# B&R Automation Studio project CamAutomat1 (part 2)

#### Main.st
```iecst
//[*********************************************************************************
//* Primary Author:    	Morteza Shahmoradi
//* Created:   			Dec 4, 2023
//* Description: 		Machine  Control
//	*********************************************************************************]
PROGRAM _INIT

	(* Initialize MpAxisBasic_AxisMaster *)
	MpAxisBasic_AxisMaster.Enable := TRUE;
	AxisParameters_Master.Position := 0.0;
	AxisParameters_Master.Velocity := 72.0;
	AxisParameters_Master.Acceleration := 3600.0;
	AxisParameters_Master.Deceleration := 3600.0;
	AxisParameters_Master.Jog.Deceleration := 3600;
	AxisParameters_Master.Stop.Deceleration := 3600.0;
	(* Initialize MpAxisBasic_AxisSlave *)
	MpAxisBasic_AxisSlave.Enable := TRUE;
	AxisParameters_Slave.Position := 0.0;
	AxisParameters_Slave.Velocity := 72.0;
	AxisParameters_Slave.Acceleration := 3600.0;
	AxisParameters_Slave.Deceleration := 3600.0;
	AxisParameters_Slave.Stop.Deceleration := 3600.0;
	AxisParameters_Slave.Jog.Deceleration := 3600;
	AxisParameters_Slave.Stop.Deceleration := 3600.0;

	AxisParameters_Master.AutoTune.Mode 				:= mcAXIS_TUNE_AUTOMATIC;
	AxisParameters_Master.AutoTune.MaxCurrentPercent 	:= 80.0;
	AxisParameters_Master.AutoTune.MaxDistance 			:= 10;
	AxisParameters_Master.AutoTune.MaxPositionError 	:= 30;

	AxisParameters_Slave.AutoTune.Mode 				:= mcAXIS_TUNE_AUTOMATIC;
	AxisParameters_Slave.AutoTune.MaxCurrentPercent 	:= 80.0;
	AxisParameters_Slave.AutoTune.MaxDistance 			:= 10;
	AxisParameters_Slave.AutoTune.MaxPositionError 	:= 30;

	MpAxisBasic_AxisMaster.MpLink := ADR(gConv_MpLink);
	MpAxisBasic_AxisMaster.Parameters := ADR(AxisParameters_Master);
	MpAxisBasic_AxisSlave.MpLink := ADR(gCutter_MpLink);
	MpAxisBasic_AxisSlave.Parameters := ADR(AxisParameters_Slave);
	MpAxisCamSequencer_0.MpLink := ADR(gCutter_MpLink);

	MpAxisCamSequencer_0.MpLinkMaster := ADR(gConv_MpLink);
	MpAxisCamSequencer_0.Parameters := ADR(CamSequencerParameters_0);

END_PROGRAM

PROGRAM _CYCLIC

	AxisParameters_Master.Velocity := gConvPrSpeed * 70 / 60 ;	// speed comes the part per minites divided by 60 s
	AxisParameters_Slave.Jog.Velocity := gCutJogSpeed;	  // Jog speed comes from HMi manaul page
	AxisParameters_Master.Jog.Velocity := gConvJogSpeed; // belt jog peed  comes from HMi manaul page
	gConvPosition := MpAxisBasic_AxisMaster.Position;  // realtime belt position  to  HMi manaul page
	gCutPosition  := MpAxisBasic_AxisSlave.Position;  // real time saw position to hmi
	gManualActive :=  NOT MpAxisBasic_AxisMaster.MoveVelocity;
	IF  (MpAxisBasic_AxisSlave.Position < cutJogEnableFWL) THEN // if the saw is not in cut zone move is backward
		AxisParameters_Slave.Direction := mcDIR_NEGATIVE;
	ELSE
		AxisParameters_Slave.Direction :=  mcDIR_POSITIVE;

	END_IF
	// Check the saw to  find where is connected
	sawInCutPosition := NOT (MpAxisBasic_AxisSlave.Position > cutJogEnableBWL AND MpAxisBasic_AxisSlave.Position < cutJogEnableFWM) AND NOT MpAxisBasic_AxisMaster.MoveVelocity ;
	displayMessageAuto := NOT sawInCutPosition AND NOT MpAxisBasic_AxisMaster.MoveVelocity ; // dispay disable message so no possibe run
	TON_DelayDo1.PT := DelayOpc;

	// Create Pulse Generator Start
	IF TON_DelayDo1.ET <> DelayOpc THEN
		TON_DelayDo1.IN := TRUE;
	END_IF
	TON_DelayDo1();
	gServoInitialized:= TON_DelayDo1.Q ;
	gDispalyServoNotReady := NOT gServoInitialized;

	// Control and Case for the Cutter and Conveyor
		CASE AxisStep OF

				STATE_WAIT :     // Wait until servo initialized  00000 ************************** STATE_WAIT ********************* 0000 ********************* STATE_WAIT
					MpAxisBasic_AxisMaster.Power		:= FALSE; // turn of drive
					MpAxisBasic_AxisSlave.Power			:= FALSE; // turn of drive Saw
					MpAxisCamSequencer_0.Enable			:= FALSE; // diale the cam sequencer
					gEnableTouchProbe := FALSE;
					IF ( Axis1.Exists AND gServoInitialized) THEN
						MpAxisBasic_AxisMaster.Power	:= TRUE;
						MpAxisBasic_AxisSlave.Power		:= TRUE;
						AxisStep :=  STATE_POWER_ON;
					END_IF

				STATE_POWER_ON : //Power on the servos **** 1 ****************** STATE_POWER_ON ********************* 1 ********************* STATE_POWER_ON
					gEnableTouchProbe := FALSE;
					IF (MpAxisBasic_AxisMaster.PowerOn = TRUE AND MpAxisBasic_AxisMaster.PowerOn = TRUE ) THEN
						AxisStep := STATE_HOME;
					END_IF
					IF (MpAxisBasic_AxisMaster.Error OR MpAxisBasic_AxisSlave.Error) THEN
						Axis1_ErrorID := 1;
						AxisStep := STATE_ERROR;
					END_IF

				STATE_HOME :  //Home the two Servo ********* 2 ********************STATE_HOME************************* 2 *********************STATE_HOME
					Axis1.statusHomed 							:= FALSE;
					AxisParameters_Master.Homing.Mode 		:= mcHOMING_DIRECT;// set the home type for the master ax
					AxisParameters_Master.Homing.Position 	:= 0.0;
					AxisParameters_Slave.Homing.Mode 		:= mcHOMING_ABSOLUTE; // set the home type abs for the slave
					AxisParameters_Slave.Homing.Position 	:= -161.4;  // relative position
					IF (NOT MpAxisCamSequencer_0.CommandBusy AND NOT MpAxisCamSequencer_0.StartSequence)  THEN
						MpAxisBasic_AxisMaster.Home 			:= TRUE;
						MpAxisBasic_AxisSlave.Home 			:= TRUE;
					END_IF

					IF EDGEPOS(MpAxisBasic_AxisMaster.IsHomed) THEN // master is homed
						Axis1Home		:= TRUE;
					END_IF

					IF EDGEPOS(MpAxisBasic_AxisSlave.IsHomed) THEN // slave is homed
						Axis2Home		:= TRUE;
					END_IF

					IF (Axis1Home AND Axis2Home) THEN  // if its home then go to ready state
						Axis1.statusHomed 			:= 1;
						MpAxisBasic_AxisMaster.Home 	:= FALSE;
						MpAxisBasic_AxisSlave.Home 	:= FALSE;
						Axis2Home := FALSE;
						Axis1Home := FALSE;
						MpAxisCamSequencer_0.Enable := TRUE;
						gEnableTouchProbe := TRUE;
						AxisStep := STATE_READY;
					END_IF
					IF (MpAxisBasic_AxisMaster.Error OR MpAxisBasic_AxisSlave.Error) THEN  // if there is an erro o to error state
						Axis1_ErrorID := 2;
						AxisStep := STATE_ERROR;
					END_IF

				STATE_READY : //Wait for the commands to change the state ***** 10 ************************ STATE_READY ******************** 10 ************************** STATE_READY
					Axis1.statusOff := 0;
					Axis1.statusStarting :=0;
					MpAxisCamSequencer_0.Enable := TRUE;
					gEnableTouchProbe := FALSE;
					CutStart := FALSE;
					disbaleHome := TRUE;	// Enable home
						// Home state if requested by HMI
					IF (Axis1.cmdHome = 1 AND NOT  MpAxisBasic_AxisMaster.CommandBusy  AND NOT  MpAxisBasic_AxisSlave.CommandBusy )THEN  // command home if
						Axis1Home							:= FALSE;
						Axis2Home							:= FALSE;
						MpAxisCamSequencer_0.StartSequence 	:= FALSE;
						AxisStep 							:= STATE_HOME;
						Axis1.cmdHome		 				:= FALSE;

					ELSIF (Axis1.cmdStop = 1) THEN  // Stop command activate from HMI

						Axis1.cmdCamAutomat 					:=FALSE;
						Axis1.cmdStop 							:= FALSE;
						Axis1.cmdMoveVelocity 					:= FALSE;
						Axis1.cmdMoveAdditive 					:= FALSE;
						MpAxisBasic_AxisMaster.MoveAdditive 	:= FALSE;
						MpAxisBasic_AxisMaster.MoveVelocity 	:= FALSE;
						AxisStep 				:= STATE_STOP;

					ELSIF MpAxisBasic_AxisMaster.MoveVelocity AND Axis1.cmdStartAutomat   THEN  // demand for the Cut
						MpAxisCamSequencer_0.StartSequence := TRUE;
						MpAxisCamSequencer_0.Signal1		:= FALSE;
						AxisStep := STATE_MOVE_CAMAUTOMAT;

					ELSIF NOT MpAxisBasic_AxisSlave.MoveAbsolute AND Axis1.cmdMoveVelocity AND NOT MpAxisBasic_AxisMaster.MoveVelocity AND  MpAxisBasic_AxisSlave.Position = 0.0  THEN
							AxisStep := STATE_MOVE_VELOCITY;
					ELSIF Axis1.cmdMoveVelocity  AND NOT (MpAxisBasic_AxisSlave.Position = 0.0  ) THEN
						MpAxisBasic_AxisSlave.MoveAbsolute := TRUE;
					ELSIF MpAxisBasic_AxisSlave.MoveAbsolute  AND  ( MpAxisBasic_AxisSlave.Position = 0.0 ) THEN
						MpAxisBasic_AxisSlave.MoveAbsolute := FALSE;
					ELSIF Axis2.cmdHome THEN
						MpAxisBasic_AxisSlave.MoveAbsolute := TRUE;
						Axis2.cmdHome := FALSE;
					ELSIF NOT MpAxisBasic_AxisMaster.MoveVelocity AND (Axis1.cmdManualForward OR Axis1.cmdManualReverse OR Axis2.cmdManualForward OR Axis2.cmdManualReverse ) THEN
						AxisStep := STATE_JOG;
						startPositionJog := MpAxisBasic_AxisMaster.Position ;
					ELSIF (Axis1.Exists = 0) THEN  // power of servos
						AxisStep := STATE_WAIT;

					END_IF

					IF MpAxisBasic_AxisMaster.Error OR MpAxisBasic_AxisSlave.Error THEN  // if there is an erro o to error state
						AxisStep := STATE_ERROR;
					END_IF

				STATE_STOP : // Stop the axis ******** 20 ****************************** STATE_STOP ***************************** 20 ********************** STATE_STOP
					Axis1.statusOff := 0;
					MpAxisBasic_AxisMaster.Stop := TRUE;
					MpAxisBasic_AxisSlave.Stop := TRUE;
					(* if axis is stopped go to state wait *)
					IF (MpAxisBasic_AxisMaster.Stopped = 1 AND MpAxisBasic_AxisSlave.Stopped = 1 ) THEN
					MpAxisBasic_AxisMaster.Stop := FALSE;
					MpAxisBasic_AxisSlave.Stop := FALSE;
						AxisStep := STATE_READY;
					END_IF
					(* check if error occured *)
					IF (MpAxisBasic_AxisMaster.Error OR MpAxisBasic_AxisSlave.Error) THEN
						Axis1_ErrorID := 3;
						AxisStep := STATE_ERROR;
					END_IF
				STATE_MOVE_ABSOLUTE : //Control Move Absolute **** 24 *************************** STATE_MOVE_ABSOLUTE *********************** 24 ******************* STATE_MOVE_ABSOLUTE

				STATE_MOVE_ADDITIVE : //Control Move Additive ** 26 *********************** STATE_MOVE_POSITION *************************** 26 ****************************STATE_MOVE_POSITION
					IF ( Axis1.cmdMoveAdditive  )	 THEN
						MpAxisBasic_AxisMaster.MoveAdditive := TRUE;
						Axis1.cmdMoveAdditive := FALSE;
						TON_StepDelay.IN			:= TRUE;
						AxisStep := STATE_READY;
					END_IF

					IF MpAxisBasic_AxisMaster.Error THEN  // if there is an erro o to error state
						AxisStep := STATE_ERROR;
					END_IF

				STATE_MOVE_VELOCITY : //Control Move velocity ** 28 *************************** STATE_MOVE_VELOCITY *********************** 28 ******************* STATE_MOVE_VELOCITY
					IF ( Axis1.cmdMoveVelocity  ) 	THEN
						MpAxisBasic_AxisMaster.MoveVelocity	:= TRUE;
						Axis1.cmdMoveVelocity := FALSE;
						AxisStep := STATE_READY;
					TON_StepDelay.IN			:= TRUE;
					Axis1.cmdStartAutomat 		:= TRUE;
					END_IF

					IF MpAxisBasic_AxisMaster.Error THEN
						AxisStep := STATE_ERROR;
					END_IF

				STATE_MOVE_CAMAUTOMAT : //Control Move automat *** 30 *************************** STATE_MOVE_VELOCITY *********************** 30 ******************* STATE_MOVE_CAMAUTOMAT
						gEnableTouchProbe := TRUE;
						MpAxisBasic_AxisMaster.Update := gSaveParameter;
						MpAxisCamSequencer_0.Signal2 := Axis1.statusOff ;
						CutStart := MpAxisCamSequencer_0.ActualStateIndex <> 0 AND enableCut;
						gEnableTouchProbe := CutStart;
					 IF NOT Axis1.cmdStartAutomat  THEN  // demand for cut activate from HMI
						Axis1.cmdCam 			:= FALSE;
						MpAxisCamSequencer_0.StartSequence 		:= FALSE;
						AxisStep := STATE_READY;
					ELSIF (Axis1.cmdStop = 1) THEN
						enableCut								:= FALSE; // Enable cut will be clear as stop cmamnd comes
						Axis1.cmdStartAutomat 					:= FALSE;
						Axis1.cmdCam 							:= FALSE;
						Axis1.cmdStop 							:= FALSE;
						Axis1.cmdMoveVelocity 					:= FALSE;
						Axis1.cmdMoveAdditive 					:= FALSE;
						MpAxisBasic_AxisMaster.MoveAdditive 	:= FALSE;
						MpAxisBasic_AxisMaster.MoveVelocity 	:= FALSE;
						MpAxisCamSequencer_0.StartSequence		:= FALSE;
						AxisStep := STATE_STOP;
					ELSIF (Axis1.statusOff = 1 AND MpAxisCamSequencer_0.ActualStateIndex = 1 ) THEN
						Axis1.cmdStartAutomat 					:= FALSE;  // production finish procedure
						Axis1.cmdCam 							:= FALSE;
						Axis1.statusOff							:= FALSE;
						Axis1.cmdMoveVelocity 					:= FALSE;
						Axis1.cmdMoveAdditive 					:= FALSE;
						MpAxisBasic_AxisMaster.MoveAdditive 	:= FALSE;
						MpAxisBasic_AxisMaster.MoveVelocity 	:= FALSE;
						MpAxisCamSequencer_0.StartSequence		:= FALSE;
						AxisStep := STATE_STOP;
						enableCut								:= FALSE;
					ELSIF MpAxisCamSequencer_0.ActualStateIndex >=1 THEN
						MpAxisCamSequencer_0.Signal1 := Axis1.cmdCam AND NOT Axis1.statusOff AND NOT twoCutEnable ;
						MpAxisCamSequencer_0.Signal2 := Axis1.cmdCam AND NOT Axis1.statusOff AND  twoCutEnable ;

					END_IF

				STATE_JOG ://************************* 40 **************************** STATE_JOG ********************************* 40 ********************* STATE_JOG

				IF NOT (Axis1.cmdManualForward OR Axis1.cmdManualReverse OR Axis2.cmdManualForward OR Axis2.cmdManualReverse ) AND  gRunPage THEN
					gRunPage := FALSE;
					AxisStep := STATE_READY;
				END_IF

				MpAxisBasic_AxisMaster.JogPositive 	:= Axis1.cmdManualForward AND sawInCutPosition; // Jog Conveyor forward
				MpAxisBasic_AxisMaster.JogNegative	:= Axis1.cmdManualReverse AND MpAxisBasic_AxisMaster.Position > (startPositionJog - 100.00) AND sawInCutPosition;
				IF 	EDGENEG(Axis1.cmdManualForward) THEN // correct the position
					startPositionJog := MpAxisBasic_AxisMaster.Position;
				END_IF
				MpAxisBasic_AxisSlave.JogPositive 	:= Axis2.cmdManualForward AND cutJogEnableFW   ;// Jog Cutter Forward
				MpAxisBasic_AxisSlave.JogNegative 	:= Axis2.cmdManualReverse AND cutJogEnableBW ; // Jog Cutter Reverse
				disbaleHome := FALSE; // disable to make zero in hmi

				STATE_ERROR : //********************** 101 ******************************* STATE_ERROR **************************** 101 ********************** STATE_ERROR
					gErrorID := 3;
					alarmActive := TRUE;
					enableCut := FALSE;
					Axis1.statusStarting :=0;
					Axis1.statusFaulted := TRUE;
					MpAxisBasic_AxisMaster.Power := FALSE;
					MpAxisBasic_AxisMaster.Home := FALSE;
					MpAxisBasic_AxisMaster.Stop := FALSE;
					MpAxisBasic_AxisMaster.MoveAbsolute := FALSE;
					MpAxisBasic_AxisMaster.MoveVelocity := FALSE;
					MpAxisBasic_AxisMaster.ErrorReset := Axis1.cmdReset;
					MpAxisBasic_AxisSlave.Power := FALSE;
					MpAxisBasic_AxisSlave.Home := FALSE;
					MpAxisBasic_AxisSlave.Stop := FALSE;
					MpAxisBasic_AxisSlave.MoveAbsolute := FALSE;
					MpAxisBasic_AxisSlave.MoveVelocity := FALSE;
					MpAxisBasic_AxisSlave.ErrorReset := Axis1.cmdReset;
					MpAxisCamSequencer_0.ErrorReset := Axis1.cmdReset;
					IF (NOT(MpAxisBasic_AxisSlave.Error ) AND NOT(MpAxisBasic_AxisMaster.Error )) THEN
						Axis1.statusFaulted:=FALSE;
						Axis1.cmdReset := FALSE;
						AxisStep := STATE_WAIT;
						Axis1.statusErrorID := 0;
						MpAxisBasic_AxisMaster.ErrorReset := FALSE;
						MpAxisBasic_AxisSlave.ErrorReset  := FALSE;
					MpAxisCamSequencer_0.ErrorReset := FALSE;
					gErrorID := 0;
					alarmActive := FALSE;

					END_IF

	END_CASE
	// Graph in the C# app
	Data[0] := MpAxisBasic_AxisMaster.Position;
	Data[1] := MpAxisBasic_AxisSlave.Position;
	Data[2] := BOOL_TO_REAL(Axis1.cmdCam) * 360.0;
	Data[3] := 0.0;
	Data[4] := 0.0;
	Data[5] := MpAxisCamSequencer_0.ActualStateIndex * 50.0;
	// Call fbs
	MpAxisBasic_AxisMaster();
	MpAxisBasic_AxisSlave();
	MpAxisCamSequencer_0();
	// Stop blade pass the cut zone
	cutJogEnableFW := (MpAxisBasic_AxisSlave.Position > -0.1  AND MpAxisBasic_AxisSlave.Position < cutJogEnableFWL ) OR // stop jog when the blade is off
	(MpAxisBasic_AxisSlave.Position > cutJogEnableFWM  AND MpAxisBasic_AxisSlave.Position < 359.9999) OR
	bypassProtection;
	cutJogEnableBW := (MpAxisBasic_AxisSlave.Position > -0.1  AND MpAxisBasic_AxisSlave.Position < cutJogEnableBWL ) OR // stop jog when the blade is off
	(MpAxisBasic_AxisSlave.Position > cutJogEnableBWM  AND MpAxisBasic_AxisSlave.Position < 359.9999) OR
	bypassProtection;

	IF gErrorID > 0 THEN  // MAchine status code
		gMachineStatus := 3; // Error
		displayStopImage := TRUE;
		displayRunImage := FALSE;
	ELSIF AxisStep = 0 AND gServoInitialized  THEN
		gMachineStatus := 6;
		displayStopImage := TRUE;
		displayRunImage := FALSE;
	ELSIF MpAxisBasic_AxisMaster.MoveVelocity AND gErrorID = 0 THEN // define the stop mode
		gMachineStatus := 1;
		displayStopImage := FALSE;
		displayRunImage := TRUE;
	ELSIF AxisStep = 40 THEN
		gMachineStatus := 2;
		displayStopImage := TRUE;
		displayRunImage := FALSE;
	ELSIF Axis1.statusOff = 1 THEN // define the stop mode finalize mpod
		gMachineStatus := 5;
		displayStopImage := TRUE;
		displayRunImage := FALSE;
	ELSIF NOT MpAxisBasic_AxisMaster.MoveVelocity AND AxisStep = 10   THEN // define the Jog mode
		gMachineStatus := 0;
		displayStopImage := TRUE;
		displayRunImage := FALSE;
	ELSIF gServoInitialized = 0 THEN // servo are intialized
		gMachineStatus := 4;
		displayStopImage := TRUE;
		displayRunImage := FALSE;
	END_IF

	gMachineStatusMessage := gMachineStatusArray[gMachineStatus];	 // HMI status
	cutEnd := (MpAxisBasic_AxisSlave.Position > cutStartDegree AND MpAxisBasic_AxisSlave.Position < cutEndDegree ) OR (MpAxisBasic_AxisSlave.Position > cutStartDegree + 180.0 AND MpAxisBasic_AxisSlave.Position < cutEndDegree +180 AND twoCutEnable );
	maxproducSpeed := maxSpeed + maxSpeed * 0.855 * twoCutEnable; // max production speed
	IF gConvPrSpeed > maxproducSpeed THEN // limit the speed to prevent fault
		gConvPrSpeed := maxproducSpeed;
	END_IF

	IF EDGEPOS(cutEnd) THEN  // if one cut done cut the signal plc
		Axis1.cmdCam := FALSE;
		cutCount := cutCount +1; // add one cut is done
	END_IF

	IF gResetCount THEN  // reset cut count
		cutCount := 0;
	END_IF

END_PROGRAM

PROGRAM _EXIT

	MpAxisBasic_AxisMaster.Enable := FALSE;
	MpAxisBasic_AxisSlave.Enable := FALSE;
	MpAxisCamSequencer_0.Enable := FALSE;
	MpAxisBasic_AxisMaster();
	MpAxisBasic_AxisSlave();
	MpAxisCamSequencer_0();

END_PROGRAM
```

### Program Logical/TouchProbe (IEC) - Save position and control trigger

#### Variables.var
```iecst
VAR
	ValidTriggerCount : UDINT; (*ValidTriggerCount comes from touch probe*)
	preValue : LREAL; (*Old position*)
	partDetected : BOOL; (*start cam*)
	newValueF : BOOL; (*New Value comes form MC BR*)
	newValue : LREAL; (*new Position*)
	MissedTriggerCount : UDINT; (*MissedTriggerCount from touch robe *)
	missedCuts : INT; (*Number of missed cuts*)
	MinWidth : LREAL := 9.0; (*MinWidth to the MC BR touchprobe, to get the valid triiger*)
	MC_BR_TouchProbe_0 : MC_BR_TouchProbe := (Period:=70,ExpectedValue:=70,WindowNegative:=20,WindowPositive:=20,Mode:=mcTP_MODE_WITHOUT_PERIOD); (*MC probe to detec the position*)
	MC_BR_ProcessParID_AcpAx_0 : MC_BR_ProcessParID_AcpAx; (*Set the battery problem Par block*)
	McBrTrigger : McBrTriggerType; (*MC Br Trigger*)
	McBrAdvancePar : McAdvBrTouchProbeParType := (ReadTriggerWidth:=1); (*MC Advance paramter*)
	McAcpAxProcessParIDPar : McAcpAxProcessParIDType := (ParID:=719,VariableAddress:=1,DataType:=mcACPAX_PARTYPE_UDINT); (*parameters*)
	MaxWidth : LREAL := 11.0; (*Maximum width for the MC triiger type - touc probe*)
	maxValueExpected : LREAL := 100.00; (*MAximum Expected Value*)
	lastAndCurrentDif : LREAL; (*last and current disatnce*)
	i : USINT; (*for saving the cuts*)
	difValue : LREAL; (*distance*)
	delatTimerProbe : TON; (*Delay for start cut*)
	cutSize : LREAL := 10.0; (*Cut Size *)
	cutDistanceAveHmi : LREAL; (*Average of last cuts to be display in hmi*)
	cutDistanceAve : LREAL; (*Average of last cuts *)
	cutDistance : ARRAY[0..7] OF LREAL; (*Lat 8 cut distance*)
	MC_BR_TouchProbe_1 : MC_BR_TouchProbe := (Period:=70,ExpectedValue:=70,WindowNegative:=20,WindowPositive:=20,Mode:=mcTP_MODE_SHIFT_FROM_RESULT); (*MC probe to detec the position*)
	McBrTrigger_1 : McBrTriggerType; (*MC Br Trigger*)
	McBrAdvancePar_1 : McAdvBrTouchProbeParType := (UseFirstTriggerPosition:=1); (*MC Advance paramter*)
	MC_BR_ProcessParID_AcpAx_1 : MC_BR_ProcessParID_AcpAx; (*Set the battery problem Par block conv*)
	currentReadingDistance : LREAL; (*Reead the current distance beween two print mark*)
END_VAR
```

#### Main.st
```iecst
//[*********************************************************************************
//* Primary Author:    	Morteza Shahmoradi
//* Created:   			Dec 7, 2023
//* Description: 		Touch Probe
//	*********************************************************************************]
PROGRAM _INIT
	(* Insert code here *)

	MC_BR_TouchProbe_1.Enable := TRUE;

END_PROGRAM

PROGRAM _CYCLIC
	// Code to write the par id 719 19, to bypass the encoder alarm, for cutter
	MC_BR_ProcessParID_AcpAx_0(Axis := ADR(gCutter_MpLink), DataAddress := ADR(McAcpAxProcessParIDPar) , NumberOfParIDs :=1 , Mode := mcACPAX_PARID_SET);
	MC_BR_ProcessParID_AcpAx_0();
	MC_BR_ProcessParID_AcpAx_1(Axis := ADR(gConv_MpLink), DataAddress := ADR(McAcpAxProcessParIDPar) , NumberOfParIDs :=1 , Mode := mcACPAX_PARID_SET);
	MC_BR_ProcessParID_AcpAx_1();

	// touch probe setup,
	MC_BR_TouchProbe_0.AdvancedParameters := McBrAdvancePar;
	MC_BR_TouchProbe_0.Axis := ADR(gConv_MpLink);
	MC_BR_TouchProbe_0.TriggerInput := McBrTrigger;
	MC_BR_TouchProbe_0();
	MC_BR_TouchProbe_0.Enable := gEnableTouchProbe;

	McBrAdvancePar.ReadTriggerWidth := TRUE; // Enable to read print lengh
	ValidTriggerCount := MC_BR_TouchProbe_0.ValidTriggerCount;// count of valid trigger
	MissedTriggerCount := MC_BR_TouchProbe_0.MissedTriggerCount; // count of missed trigger
	MC_BR_TouchProbe_0.TriggerInput.MaxWidth := MaxWidth; // MaxWidth to the touch probe
	MC_BR_TouchProbe_0.TriggerInput.MinWidth := MinWidth; // Min Width to the touch rpobe

	// second touch probe for training purpose
	MC_BR_TouchProbe_1.AdvancedParameters := McBrAdvancePar_1;
	MC_BR_TouchProbe_1.Axis := ADR(gConv_MpLink);
	MC_BR_TouchProbe_1.TriggerInput := McBrTrigger_1;
	MC_BR_TouchProbe_1();
	MC_BR_TouchProbe_1.Enable := NOT gResetCount;

	currentReadingDistance := MC_BR_TouchProbe_1.Period - MC_BR_TouchProbe_1.DeltaExpectedValue;

	// manaul paramter find

	newValue := MC_BR_TouchProbe_0.RecordedValue;
	IF newValue > ( preValue + cutSize) THEN  // check if its a new print mark coms
		difValue := newValue - preValue ;  // calculates
		IF difValue > gMinValue THEN   // validate correct distance
			newValueF := TRUE;
			preValue := newValue;
			partDetected := delatTimerProbe.Q ; // part is detected rise cut flag
			IF difValue < maxValueExpected THEN
				FOR i := 0 TO 6 BY 1 DO
					cutDistance[7-i] := cutDistance[6-i] ;
				END_FOR
				cutDistance [0] := difValue;
				lastAndCurrentDif := difValue; // for Hmi display
				cutDistanceAve := 0;
				FOR i := 0 TO 7 BY 1 DO			// save old data
					cutDistanceAve := cutDistanceAve + cutDistance[i] ;
				END_FOR
				cutDistanceAveHmi := cutDistanceAve/ 8;
			END_IF
		END_IF

		IF difValue < gMinValue AND newValueF THEN   // count missed cuts
			missedCuts := missedCuts + 1;
			newValueF := FALSE;
		END_IF

	END_IF

	IF gResetCount THEN  // reset cut count
		missedCuts := 0;
		gResetCount := FALSE;
	END_IF

	delatTimerProbe(IN := CutStart , PT := T#500ms);
	delatTimerProbe();
	IF 	EDGEPOS(partDetected) AND delatTimerProbe.Q  THEN // activate the cut when the touch is 70mm after that
		Axis1.cmdCam := TRUE;
		partDetected := FALSE;
	END_IF

	IF EDGEPOS(Axis1.cmdStartAutomat) THEN // transfer the cut last and new position to the last position
		preValue := newValue;
	END_IF
	IF EDGEPOS(gEnableTouchProbe) THEN  // reset the partDetected bit to prevent stop in jog
		partDetected := FALSE;
	END_IF

	//  get paramter infor from cam automat

END_PROGRAM

PROGRAM _EXIT
	(* Insert code here *)
	MC_BR_TouchProbe_0.Enable := FALSE;
	MC_BR_TouchProbe_0();
	MC_BR_TouchProbe_1.Enable := FALSE;
	MC_BR_TouchProbe_1();

END_PROGRAM
```

### Program Logical/MachineAlarm (IEC) - Alarm Control

#### Variables.var
```iecst
VAR
	MpAlarmXCore_0 : MpAlarmXCore; (*mp alarm core x function block *)
	MpAlarmXAcknowledgeAll_0 : MpAlarmXAcknowledgeAll; (*Reset alarm list*)
	ackAlarms : BOOL; (*Hmi request to delete alarm*)
END_VAR
```

#### Main.st
```iecst
//[*********************************************************************************
//* Primary Author:    	Morteza Shahmoradi
//* Created:   			Dec 7, 2023
//* Description: 		Machine  Alarm
//	*********************************************************************************]
PROGRAM _INIT
	(* Insert code here *)
	MpAlarmXCore_0(
				MpLink := ADR(MpLinkMachinegAlarmXCore),
				Enable := TRUE, );
	//		ErrorReset := );
	MpAlarmXAcknowledgeAll_0(
	MpLink := ADR(MpLinkMachinegAlarmXCore),
	Enable := TRUE, );
	//		ErrorReset := );
END_PROGRAM

PROGRAM _CYCLIC

	MpAlarmXCore_0();

	MpAlarmXAcknowledgeAll_0.Execute := ackAlarms;
	MpAlarmXAcknowledgeAll_0();
	ackAlarms := FALSE;

END_PROGRAM

PROGRAM _EXIT
	(* Insert code here *)

	MpAlarmXCore_0.Enable:= FALSE;
	MpAlarmXCore_0();
	MpAlarmXAcknowledgeAll_0.Enable:= FALSE;
	MpAlarmXAcknowledgeAll_0();
END_PROGRAM
```

### Program Logical/RecipeMgmt (IEC) - Manage Recipe

#### Cyclic.ld - Cyclic code
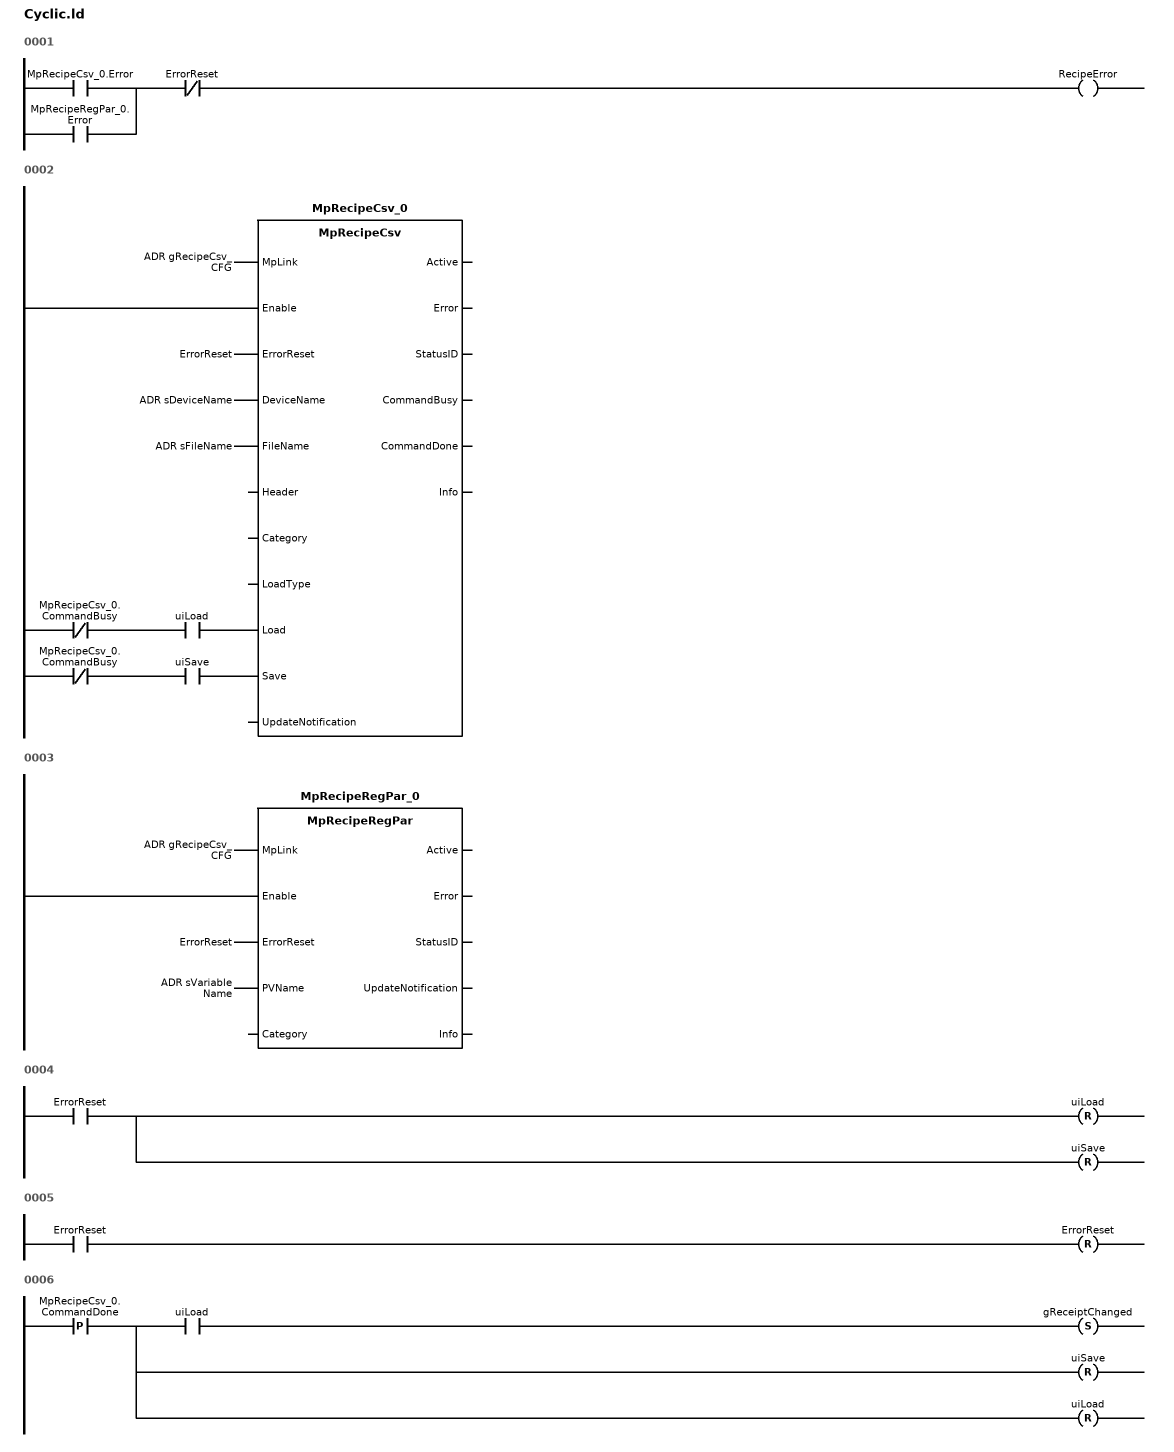
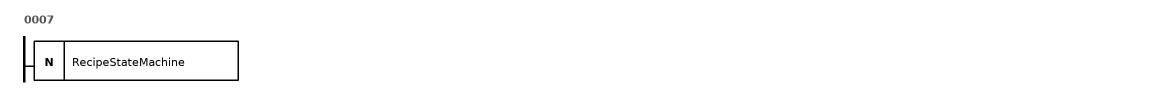
Ladder, written as Structured Text:
```iecst
PROGRAM _CYCLIC
VAR
    _e1 : R_TRIG;
END_VAR
(* Network 1 *)
RecipeError := (MpRecipeCsv_0.Error OR MpRecipeRegPar_0.Error) AND NOT ErrorReset;

(* Network 2 *)
MpRecipeCsv_0(MpLink := ADR(gRecipeCsv_CFG), Enable := TRUE, ErrorReset := ErrorReset, DeviceName := ADR(sDeviceName), FileName := ADR(sFileName), Load := NOT MpRecipeCsv_0.CommandBusy AND uiLoad, Save := NOT MpRecipeCsv_0.CommandBusy AND uiSave);

(* Network 3 *)
MpRecipeRegPar_0(MpLink := ADR(gRecipeCsv_CFG), Enable := TRUE, ErrorReset := ErrorReset, PVName := ADR(sVariableName));

(* Network 4 *)
IF ErrorReset THEN
    uiLoad := FALSE;
    uiSave := FALSE;
END_IF;

(* Network 5 *)
IF ErrorReset THEN ErrorReset := FALSE; END_IF;

(* Network 6 *)
_e1(CLK := MpRecipeCsv_0.CommandDone);
IF _e1.Q AND uiLoad THEN gReceiptChanged := TRUE; END_IF;
IF _e1.Q THEN
    uiSave := FALSE;
    uiLoad := FALSE;
END_IF;

(* Network 7 *)
RecipeStateMachine;
END_PROGRAM
```

#### Init.ld - Initialization code
Ladder, written as Structured Text:
```iecst
PROGRAM _INIT
END_PROGRAM
```

#### Exit.ld - Exit code
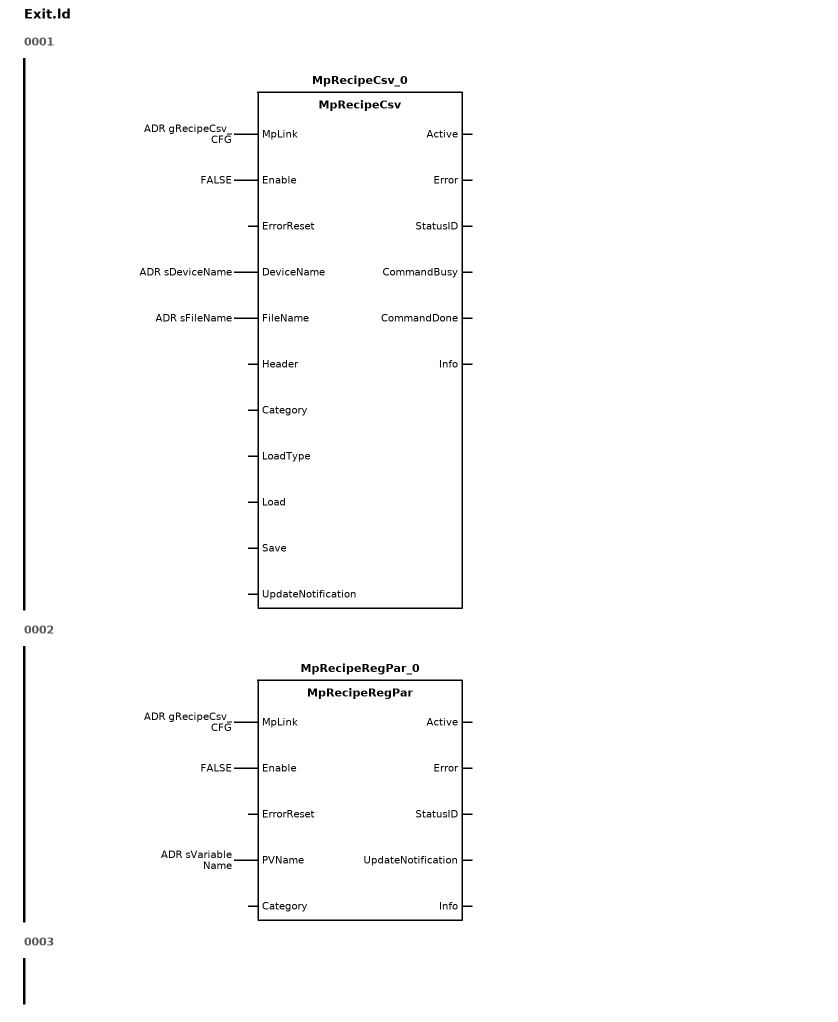
Ladder, written as Structured Text:
```iecst
PROGRAM _EXIT
(* Network 1 *)
MpRecipeCsv_0(MpLink := ADR(gRecipeCsv_CFG), Enable := FALSE, DeviceName := ADR(sDeviceName), FileName := ADR(sFileName));

(* Network 2 *)
MpRecipeRegPar_0(MpLink := ADR(gRecipeCsv_CFG), Enable := FALSE, PVName := ADR(sVariableName));

(* Network 3 *)
END_PROGRAM
```

#### Types.typ - Local data types
```iecst
TYPE
	State_enum :
		(
		WAIT,
		SAVE,
		LOAD
		);
END_TYPE
```

#### Variables.var - Local variables
```iecst
VAR
	uiLoad : BOOL := FALSE; (*Hmi demand to load*)
	uiSave : BOOL; (*Hmi demand to save data to plc harddisk*)
	sDeviceName : STRING[255] := 'CSV_Recipes'; (*device name (set in the cpu configuration)*)
	sFileName : STRING[255] := 'recipe1'; (*NAme of the saved file*)
	sVariableName : STRING[255] := 'gCutPar'; (*name of the variable to be saved in the PLC*)
	MpRecipeCsv_0 : MpRecipeCsv; (*mp recepie fucntion block*)
	MpRecipeRegPar_0 : MpRecipeRegPar; (*function block parameter*)
	RecipeError : BOOL; (*if there is an error*)
	ErrorReset : BOOL;
END_VAR
VAR RETAIN
	RecipeCurrent : STRING[100]; (*Current recipe*)
END_VAR
VAR
	DataProviderMid : ARRAY[0..2] OF STRING[90]; (*Data Provider*)
END_VAR
VAR RETAIN
	DataProvider : ARRAY[0..2] OF STRING[100]; (*Data Provider*)
	RecipeList : ARRAY[0..2] OF STRING[65]; (*List of recepie*)
END_VAR
VAR
	DataProviderTail : ARRAY[0..2] OF STRING[25] := ['{"value":"0","text":"','{"value":"1","text":"','{"value":"2","text":"']; (*Data Provider*)
	DataProviderHead : ARRAY[0..2] OF STRING[10] := [3('"}')]; (*Data Provider*)
	i : INT; (*to be used at for and while loop*)
	MC_BR_CamAutomatGetPar_AcpAx_0 : MC_BR_CamAutomatGetPar_AcpAx := (Command:=mcSET_ALL_PAR_FROM_ADR,CamAutomat:=(DataObjectName:='Feature_CamAutomat')); (*Get parameter from cam automat*)
	MC_BR_CamAutomatSetPar_AcpAx_0 : MC_BR_CamAutomatSetPar_AcpAx := (Command:=mcSET_ALL_PAR_FROM_ADR,CamAutomat:=(DataObjectName:='Feature_CamAutomat')); (*Set Parameters CAM ID*)
	McAcpAxAdvCamAutSetPar : McAcpAxAdvCamAutSetParType; (*Command for the transfer of the parameter
*)
	McAcpAxCamAutDefinetyp : McAcpAxCamAutDefineType := (DataObjectName:='Feature_CamAutomat'); (*Command for the transfer of the parameter
*)
END_VAR
VAR RETAIN
	McAcpAxCamAutPartypDef : ARRAY[0..2] OF McAcpAxCamAutParType; (*Command for the transfer of the parameter Current Defaults
*)
	McAcpAxCamAutPartyp : McAcpAxCamAutParType; (*Command for the transfer of the parameter Current
*)
END_VAR
VAR
	CutType : UDINT := 1; (*Cut Type *)
	copyAll : BOOL; (*Copy all partameter *)
	copySelction : BOOL := TRUE; (*Copy selection to the memory*)
	upperPosition : LREAL := 8; (*Upper Position*)
	lowerPosition : LREAL := 10; (*Lower cut Position*)
	pasteSelection : BOOL; (*Paste form default*)
	copySelctionValid : BOOL; (*Copy Valid Data to selection*)
	MS_TEST_BIT0 : BOOL := TRUE; (*Test bit to find the bug for set paramters*)
	selectedCutType : STRING[100] := 'Loading Cut Type ....'; (*selected cut type*)
	cutTypeDefault : ARRAY[0..2] OF STRING[100] := ['Middle Cut','Upper Edge Cut','Lower Edge Cut']; (*default cut types*)
END_VAR
```

#### RecipeStateMachine.st - Manage Recepie
```iecst
//[*********************************************************************************
//* Primary Author:    	Morteza Shahmoradi
//* Created:   			Dec 7, 2023
//* Description: 		recpie management
//	*********************************************************************************]
ACTION RecipeStateMachine:

	McAcpAxCamAutDefinetyp.DataAddress := ADR(McAcpAxCamAutPartyp);
	MC_BR_CamAutomatGetPar_AcpAx_0(Slave := ADR(gCutter_MpLink) , CamAutomat := McAcpAxCamAutDefinetyp);

	MC_BR_CamAutomatSetPar_AcpAx_0(Slave := ADR(gCutter_MpLink) , CamAutomat := McAcpAxCamAutDefinetyp , AdvancedParameters := McAcpAxAdvCamAutSetPar);

	IF  gReceiptChanged THEN // Recepit Change paramter command comes from HMI

		RecipeCurrent := gCutPar[gRecepitRefHmi].RecipeName;
		CutType	:= gCutPar[gRecepitRefHmi].selCutType;
		gMinValue := gCutPar[gRecepitRefHmi].minimumCutSpped;
		gConvPrSpeed := gCutPar[gRecepitRefHmi].productionSpeed;
		upperPosition :=  gCutPar[gRecepitRefHmi].upperPosition;
		lowerPosition := gCutPar[gRecepitRefHmi].lowerPosition;
		FOR i := 0 TO 2 BY 1 DO
			RecipeList[i] := gCutPar[i].RecipeName;
		END_FOR;
		pasteSelection := TRUE;  // Ececute of cam automat save

		gReceiptChanged := FALSE;
	END_IF

	IF gSaveParameter THEN  // save paramter command comes from HMI
		gCutPar[gRecepitRefHmi].RecipeName := RecipeCurrent;
		RecipeList [gRecepitRefHmi] := RecipeCurrent;
		gCutPar[gRecepitRefHmi].selCutType := CutType;
		gCutPar[gRecepitRefHmi].upperPosition := upperPosition;
		gCutPar[gRecepitRefHmi].lowerPosition := lowerPosition;
		gCutPar[gRecepitRefHmi].minimumCutSpped := gMinValue;
		gCutPar[gRecepitRefHmi].productionSpeed := gConvPrSpeed;

		gSaveParameter := FALSE; // Ececute of cam automat save
		copySelctionValid := TRUE;

	END_IF
	IF 	EDGEPOS( MC_BR_CamAutomatSetPar_AcpAx_0.Done) THEN // remove the excute command after save
		MC_BR_CamAutomatSetPar_AcpAx_0.Execute := FALSE;
	END_IF

		FOR i := 0 TO 2 BY 1 DO  // create data provider for recepir selection
		DataProviderMid[i] := CONCAT(DataProviderTail[i],RecipeList[i]);
		DataProvider[i] := CONCAT(DataProviderMid[i],DataProviderHead[i]);
	END_FOR;

	IF copyAll THEN
		gCutPar[1] := gCutPar[0] ;
		gCutPar[2] := gCutPar[0] ;

	END_IF
	IF EDGEPOS(gServoInitialized) THEN  // need to load good paramters
		uiLoad := TRUE;
	END_IF

		MC_BR_CamAutomatGetPar_AcpAx_0.Execute := copySelction AND gManualActive AND NOT gSaveParameter  AND NOT gReceiptChanged AND gServoInitialized AND NOT gvalidDateCamExist ;
	IF MC_BR_CamAutomatGetPar_AcpAx_0.Done THEN  // copy paramters to the data
		copySelction := FALSE;
		MC_BR_CamAutomatGetPar_AcpAx_0.Execute := FALSE; // get the right paramter at the start up
		McAcpAxCamAutPartypDef[0]:= McAcpAxCamAutPartyp;
		McAcpAxCamAutPartypDef[1]:= McAcpAxCamAutPartyp;
		McAcpAxCamAutPartypDef[2]:= McAcpAxCamAutPartyp; // save the parater to the diffrent set up
		McAcpAxCamAutPartypDef[1].State[2].CompensationParameters.SlaveCompDistance := McAcpAxCamAutPartypDef[0].State[2].CompensationParameters.SlaveCompDistance - upperPosition;
		McAcpAxCamAutPartypDef[1].State[4].CompensationParameters.SlaveCompDistance := McAcpAxCamAutPartypDef[0].State[4].CompensationParameters.SlaveCompDistance + upperPosition;
		McAcpAxCamAutPartypDef[1].State[5].CompensationParameters.SlaveCompDistance := McAcpAxCamAutPartypDef[0].State[5].CompensationParameters.SlaveCompDistance - upperPosition;
		McAcpAxCamAutPartypDef[1].State[7].CompensationParameters.SlaveCompDistance := McAcpAxCamAutPartypDef[0].State[7].CompensationParameters.SlaveCompDistance + upperPosition;

		McAcpAxCamAutPartypDef[2].State[2].CompensationParameters.SlaveCompDistance := McAcpAxCamAutPartypDef[0].State[2].CompensationParameters.SlaveCompDistance + lowerPosition;
		McAcpAxCamAutPartypDef[2].State[4].CompensationParameters.SlaveCompDistance := McAcpAxCamAutPartypDef[0].State[4].CompensationParameters.SlaveCompDistance - lowerPosition;
		McAcpAxCamAutPartypDef[2].State[5].CompensationParameters.SlaveCompDistance := McAcpAxCamAutPartypDef[0].State[5].CompensationParameters.SlaveCompDistance + lowerPosition;
		McAcpAxCamAutPartypDef[2].State[7].CompensationParameters.SlaveCompDistance := McAcpAxCamAutPartypDef[0].State[7].CompensationParameters.SlaveCompDistance - lowerPosition;
		pasteSelection := TRUE;
		gvalidDateCamExist := TRUE;
	END_IF

	IF copySelctionValid AND gvalidDateCamExist THEN // if the valid datat esit then adjust the state of the machine
		McAcpAxCamAutPartypDef[1].State[2].CompensationParameters.SlaveCompDistance := McAcpAxCamAutPartypDef[0].State[2].CompensationParameters.SlaveCompDistance - upperPosition;
		McAcpAxCamAutPartypDef[1].State[4].CompensationParameters.SlaveCompDistance := McAcpAxCamAutPartypDef[0].State[4].CompensationParameters.SlaveCompDistance + upperPosition;
		McAcpAxCamAutPartypDef[1].State[5].CompensationParameters.SlaveCompDistance := McAcpAxCamAutPartypDef[0].State[5].CompensationParameters.SlaveCompDistance - upperPosition;
		McAcpAxCamAutPartypDef[1].State[7].CompensationParameters.SlaveCompDistance := McAcpAxCamAutPartypDef[0].State[7].CompensationParameters.SlaveCompDistance + upperPosition;

		McAcpAxCamAutPartypDef[2].State[2].CompensationParameters.SlaveCompDistance := McAcpAxCamAutPartypDef[0].State[2].CompensationParameters.SlaveCompDistance + lowerPosition;
		McAcpAxCamAutPartypDef[2].State[4].CompensationParameters.SlaveCompDistance := McAcpAxCamAutPartypDef[0].State[4].CompensationParameters.SlaveCompDistance - lowerPosition;
		McAcpAxCamAutPartypDef[2].State[5].CompensationParameters.SlaveCompDistance := McAcpAxCamAutPartypDef[0].State[5].CompensationParameters.SlaveCompDistance + lowerPosition;
		McAcpAxCamAutPartypDef[2].State[7].CompensationParameters.SlaveCompDistance := McAcpAxCamAutPartypDef[0].State[7].CompensationParameters.SlaveCompDistance - lowerPosition;
		pasteSelection := TRUE; // set the parameter to the servos
	END_IF

	IF pasteSelection AND NOT gSaveParameter  AND NOT gReceiptChanged AND gvalidDateCamExist AND NOT uiLoad THEN // only save the new cam dat if its valid

		McAcpAxCamAutPartyp :=  McAcpAxCamAutPartypDef[CutType-1]; // cam data is valid copy
		MC_BR_CamAutomatSetPar_AcpAx_0.Execute := pasteSelection AND gManualActive AND MS_TEST_BIT0 ;
		pasteSelection := FALSE;
		selectedCutType := cutTypeDefault[gCutPar[gRecepitRefHmi].selCutType-1];

	END_IF

END_ACTION
```

- Project.language - Project Language (not shown)

### Program Logical/Recipe (IEC)

#### Cyclic.st - Cyclic code
```iecst
PROGRAM _CYCLIC
	(* Insert code here *)

END_PROGRAM
```

### Program Logical/SesnorSim

#### Main.st
```iecst
//[*********************************************************************************
//* Primary Author:    	Morteza Shahmoradi
//* Created:   			Dec 4, 2023
//* Description: 		Machine  Control
//	*********************************************************************************]
PROGRAM _INIT
	(* Insert code here *)

END_PROGRAM

PROGRAM _CYCLIC
	(* Insert code here *)

	IF  0.0 < Data[0] AND Data[0] < 10.0 THEN	/// Simulation gSensorUpStream every 50degree one whole
		gSensorUpStream := TRUE;
	ELSE
		gSensorUpStream := FALSE;
	END_IF
	Data[3] := gSensorUpStream * 360.0;

	IF  145.0 < Data[0] AND Data[0] < 155.0 AND  Data[1] > 175.0 AND Data[1] < 185.0 THEN	 /// Simulation gSensorLowStream
		gSensorLowStream := TRUE;
	ELSE
		gSensorLowStream := FALSE;
	END_IF

	Data[4] := gSensorLowStream * 360.0;

//	IF 	EDGEPOS(gSensorUpStream) AND CutStart THEN
//		Axis1.cmdCam := TRUE;
//	END_IF
//

END_PROGRAM

PROGRAM _EXIT
	(* Insert code here *)

END_PROGRAM
```

Listed in the project but not available here: Logical/Libraries/ComTCP/ComTCP_P, Logical/Recipe/Init.st, Logical/Recipe/Exit.st, Logical/Recipe/Types.typ, Logical/Recipe/Variables.var
